Yaskawa INFORM job: WELDING-FRONT-ST-2.JBI

/JOB
//NAME WELDING-FRONT-ST-2
//POS
///NPOS 0,0,0,0,0,0
//INST
///DATE 2018/11/28 18:06
///ATTR SC,RW
NOP
SETREG MREG#(112) 2
'***** CMF 100 sensor
IFTHEN D005=8
	 CALL JOB:WELDING-CMF100-ST2-FRONT
ENDIF
'***** F........ sensors
IFTHEN D005=4
	 CALL JOB:WELDING-F-SENSORS-FRONT-ST2
ENDIF
END
